FUNCTION_BLOCK DisjuntorCAT (* Composite Function Block Type *)
  (* Standard: 61499-2 *)
  (* Version 0.0, 19/05/2026, template *)
  PACKAGE Hidryco.HidrycoLib;
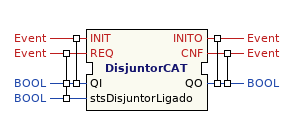
  EVENT_INPUT
    INIT WITH QI; (* Initialization Request *)
    REQ WITH QI, stsDisjuntorLigado; (* Normal Execution Request *)
  END_EVENT
  EVENT_OUTPUT
    INITO WITH QO; (* Initialization Confirm *)
    CNF WITH QO; (* Execution Confirmation *)
  END_EVENT
  VAR_INPUT
    QI : BOOL; (* Input event qualifier *)
    stsDisjuntorLigado : BOOL;
  END_VAR
  VAR_OUTPUT
    QO : BOOL; (* Output event qualifier *)
  END_VAR
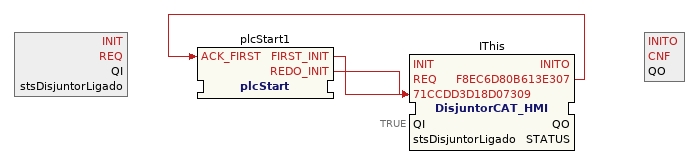
  FBS
    IThis : DisjuntorCAT_HMI(QI := TRUE);
    plcStart1 : plcStart;
  END_FBS
  EVENT_CONNECTIONS
    plcStart1.FIRST_INIT TO IThis.71CCDD3D18D07309;
    plcStart1.REDO_INIT TO IThis.71CCDD3D18D07309;
    IThis.F8EC6D80B613E307 TO plcStart1.ACK_FIRST;
  END_CONNECTIONS
END_FUNCTION_BLOCK
